(* CODESYS project 20_CS3_SQL

Project tree, tasks and I/O mapping:
  CC000xxx : 751-9401 WAGO Compact Controller 100, WAGO, order no. 751-9401, version 6.3.1.5
    application Application
      libraries: WagoSolSolutionBuilder, 1.0.0.5 (WAGO)
      task Task (cyclic, interval t#50ms, priority 15) calls PLC_PRG
      Application Template/
        ApplicationTemplateManager
          ApplicationParameters
        global variables GVL_ApplicationParameters
        program PrgRecipeHandling [ST]
        RecipeManager
          recipe definition ApplicationParameters: bLedBlinkCount : BYTE; bLedBlinkVelocity : BYTE
        text list TemplateManagerTextList
      program PLC_PRG [ST]
    Compact_Controller_100_Onboard_IO : Compact Controller 100 Onboard IO, WAGO, version 0.0.1.4
        output Application.PLC_PRG.xWD : BOOL  // X5.DO.X5.DO3
        output Application.PLC_PRG.xWD_ : BOOL  // X5.DO.X5.DO4
        unmapped channels: X12.DI, X13.PT1+/X13.PT1-, X13.PT2+/X13.PT2-, X14.AI1, X14.AI2, X5.DO, X6.AO1, X6.AO2
    Serial
      COM1 : COM1, WAGO, version 0.0.0.19
  PFC000xxx : 750-8212 PFC200, WAGO, order no. 750-8212, version 6.4.6.10
    application Application
      libraries: WagoAppRunningText, 0.0.0.1 (WAGO); WagoAppAppLED, 1.7.2.2 (WAGO); WagoSolSolutionBuilder, 1.0.0.5 (WAGO); VisuDialogs, * (System); WagoAppSQL_MySQL, 1.6.2.6 (WAGO); WagoSysErrorBase, 1.6.2.6 (WAGO); WagoSysSQLite_FR, 1.0.8.0 (WAGO_FR)
      task Task (cyclic, interval t#50ms, priority 15) calls PLC_PRG
      task TrendRecordingTask (cyclic, interval 100 ms, priority 15) calls VisuTrendStorageAccess.GlobalInstances.g_TrendRecordingManager.CyclicCall
      task VISU_TASK (cyclic, interval 100 ms, priority 15) calls VisuElems.Visu_Prg
      Application Template/
        global variables ApplicationParameters
        ApplicationTemplateManager
          ApplicationParameters
        program PrgRecipeHandling [ST]
        RecipeManager
          recipe definition ApplicationParameters: ApplicationParameters.sRunningText : STRING; ApplicationParameters.tBlinkTime01 : TIME; ApplicationParameters.tBlinkTime02 : TIME; ApplicationParameters.tBlinkTime03 : TIME; ApplicationParameters.wFunctionSelector : WORD
        text list TemplateManagerTextList
      global variables gvl_AppData
      MySQL/
      program PLC_PRG [ST]
      program PRG_MySQL [ST]
      program PRG_SQlite [ST]
      visualisation SigTrendlog
      SQlite/
      Trend Recording Manager
        SigTrendlog_Trend
      data type typSQlite_TableTest
      visualisation WSB_Example
    Kbus : Kbus, WAGO, version 2.1.0.1
        unmapped channels: K-BUS diagnostics
      _75x_16DO_1 : 75x-16DO, WAGO, version 2.0.0.13
          output wTrm1 : WORD  // _OUT
      _75x_16DO_2 : 75x-16DO, WAGO, version 2.0.0.13
          output wTrm2 : WORD  // _OUT
      _75x_16DO_3 : 75x-16DO, WAGO, version 2.0.0.13
          output wTrm3 : WORD  // _OUT
      _75x_4DI_1 : 75x-4DI, WAGO, version 2.0.0.13
          unmapped channels: _IN
    Serial
      COM1 : COM1, WAGO, version 0.0.0.19
  libraries: VisuSymbols, 4.4.0.0 (System); WagoVisuIcons, 1.1.0.8 (WAGO); WagoVisuIconsMaterialDesign, 1.0.0.2 (WAGO)
  text list GlobalTextList
*)

// PFC000xxx/Application/typSQlite_TableTest
TYPE typSQlite_TableTest :
STRUCT
	iValue			: INT;
	rValue			: REAL;
	sValue			: STRING;
	xValue			: BOOL;
END_STRUCT
END_TYPE

// PFC000xxx/Application/gvl_AppData
{attribute 'qualified_only'}
VAR_GLOBAL
	g_rSignal_SINUS				: REAL;
	g_rSignal_COSINUS			: REAL;
	g_rSignal_TRIANGLE			: REAL;
	g_rSignal_SAW				: REAL;
END_VAR

// CC000xxx/Application/Application Template/GVL_ApplicationParameters
//{attribute 'qualified_only'}
VAR_GLOBAL
	bLedBlinkCount 			: BYTE	:= 2;
	bLedBlinkVelocity 		: BYTE	:= 3;
END_VAR

// PFC000xxx/Application/Application Template/ApplicationParameters
{attribute 'qualified_only'}
VAR_GLOBAL
	// Application Parameter 1
	sRunningText: STRING := '1';
	// Application Parameter 2
	tBlinkTime01: TIME;
	// Application Parameter 3
	tBlinkTime02: TIME;
	// Application Parameter 4
	tBlinkTime03: TIME;
	// Application Parameter 5
	wFunctionSelector : WORD;		
END_VAR

// CC000xxx/Application/PLC_PRG
PROGRAM PLC_PRG
VAR
	(* cycle counter *)
	uiCnt						: UINT;
	xWD							: BOOL;
	xWD_						: BOOL;
	
END_VAR

(* cycle counter *)
uiCnt := uiCnt + 1;
xWD := uiCnt.3;
xWD_ := NOT xWD;

END_PROGRAM

// PFC000xxx/Application/PLC_PRG
PROGRAM PLC_PRG
(* **************************************************************************************** *)
(* * PROJECT INFORMATION																	*)
(* *********+***********************+****************************************************** *)
(* Author:  ¦ Stephane Rey			¦ plc acces: admin / ...								*)
(* Date:	¦ 01.07.25				¦ IP-address: 172.16.250.x/24 (dhcp)					*)
(* Version:	¦ V04.01.02.00			¦ IP-address (VPN):	10.235.0.2							*)
(* *********+*******+***************+****************************************************** *)
(* version history	¦				¦														*)
(* 01.07.25			¦ V04.01.02.00	¦ fist version											*)
(* 					¦ 				¦ CS3.5.19.07											*)
(* 					¦ 				¦														*)
(* *****************+***************+****************************************************** *)
VAR
	(* cycle counter *)
	uiCnt						: UINT;
	
	(* running text *)
	oRunningText				: WagoAppRunningText.FbRunningText;
	tRunningTextSpeed			: TIME := T#20MS;
	aRunningTextOut				: WagoAppRunningText.WLS_OUTPUTS;
	
	(* LED driver *)
	bFunctionSelectorOut		: BYTE;		
	oTOF_1						: TOF;
	oLED01						: FbAppLED_SetStatic;
	xLED01_Enable				: BOOL;
	xLED01_Error				: BOOL;
	xLED01_Valid				: BOOL;
	xLED01_Busy					: BOOL;
	oLED01_FbResult				: WagoAppAppLED.FbResult;
	eLedColor01					: WagoAppAppLED.WagoTypesAppLED.eLedColor;
	eLedColor01_				: WagoAppAppLED.WagoTypesAppLED.eLedColor;
	uiLedCount					: UINT;
	
	(* recipe management *)
	xRecipe_Read				: BOOL;
	xRecipe_Write				: BOOL;
	xRecipe_Ready				: BOOL;
	xRecipe_Busy				: BOOL;
END_VAR

(* cycle counter *)
{region 'plc-cycle-counter'}
	uiCnt := uiCnt + 1;
{endregion}

(* running text *)
{region 'running-text'}
	oRunningText(	tSpeed:= tRunningTextSpeed, 
					sText:= ApplicationParameters.sRunningText, 
					Outputs:= aRunningTextOut);
	
	(* asseign data to ourput terminals *)			
	wTrm1 := aRunningTextOut[1];	//750-1504
	wTrm2 := aRunningTextOut[2];	//750-1504
	wTrm3 := aRunningTextOut[3];	//750-1504
{endregion}

(* LED driver *)
{region 'led-driver'}
	// app selector
	CASE ApplicationParameters.wFunctionSelector OF		
		0:	// LED off
			eLedColor01:=WagoAppAppLED.WagoTypesAppLED.eLedColor.Off;
		
		1:	// LED blink yellow, sequence 1
			oTOF_1(IN:=NOT oTOF_1.Q , PT:=ApplicationParameters.tBlinkTime01);
			IF NOT oTOF_1.Q THEN
				bFunctionSelectorOut:=bFunctionSelectorOut+1;
			END_IF
			eLedColor01:=WagoAppAppLED.WagoTypesAppLED.eLedColor.Yellow;
			
		2:	// LED blink green, sequence 2
			oTOF_1(IN:=NOT oTOF_1.Q , PT:=ApplicationParameters.tBlinkTime02 );
			IF NOT oTOF_1.Q THEN
				bFunctionSelectorOut:=bFunctionSelectorOut*2;
				IF bFunctionSelectorOut=0 THEN
					bFunctionSelectorOut:=1;
				END_IF
			END_IF
			eLedColor01:=WagoAppAppLED.WagoTypesAppLED.eLedColor.Green;
			
		3:	// LED blink red, sequence 3
			oTOF_1(IN:=NOT oTOF_1.Q , PT:=ApplicationParameters.tBlinkTime03 );
			IF NOT oTOF_1.Q THEN
				bFunctionSelectorOut:=NOT bFunctionSelectorOut;
			END_IF
			eLedColor01:=WagoAppAppLED.WagoTypesAppLED.eLedColor.Red;
		ELSE
			ApplicationParameters.wFunctionSelector := 0;
	END_CASE
	
	//write new sequence management
	IF eLedColor01 <> eLedColor01_ THEN
		xLED01_Enable:=FALSE;
		uiLedCount:=uiLedCount+1;
		IF uiLedCount>10 THEN
			xLED01_Enable:=TRUE;
			eLedColor01_:=eLedColor01;
			uiLedCount:=0;
		END_IF
	END_IF
	
	// call LED driver
	oLED01(
		oStatus	=>oLED01_FbResult, 
		xEnable		:=xLED01_Enable, 
		xError		=>xLED01_Error, 
		xValid		=>xLED01_Valid, 
		xBusy		=>xLED01_Busy, 
		eLedID		:=WagoAppAppLED.eLedID.AppLED_1, 
		eLedColor	:=eLedColor01);
{endregion}	

(* recipe management *)
{region 'recipe-mngt'}
	PrgRecipeHandling(xRead:= xRecipe_Read, xWrite:= xRecipe_Write, xRecipeReady=> xRecipe_Ready, xBusy=> xRecipe_Busy);
{endregion}
	
(* application *)
{region 'application'}
	PRG_MySQL();
	PRG_SQlite();
	//ca l'air de fonctionner
{endregion}

END_PROGRAM

// CC000xxx/Application/Application Template/PrgRecipeHandling
//Program to handle the recipe parameters of the application
//{error 'Veuillez appeler ce programme dans votre programme principal ou dans une tâche pour l'activer. Supprimez ensuite cette ligne.'}
PROGRAM PrgRecipeHandling
VAR_INPUT
	xRead	: BOOL;	//Read parameters from recipe to application. (also done by tCycleTime)
	xWrite	: BOOL;	//Write parameters from application to recipe.
END_VAR
VAR_OUTPUT
	xRecipeReady	: BOOL;	//Outputs recipe parameters are ready to use in application
END_VAR
VAR
	FbRecipeApplicationParameters	: WagoSolSolutionBuilder.FbRecipeManagement;
	sApplicationParameters			: STRING:='ApplicationParameters';	//Name of the recipe definition.
	oStatusRecipeApplicationParameters	: WagoSolSolutionBuilder.WagoSysErrorBase.FbResult;
END_VAR

//call recipe manager with recipe definiction name "ApplicationParameters"
FbRecipeApplicationParameters(
	sRecipeDefinition	:= sApplicationParameters,
	tCycleTime			:= T#10S,
	xRead				:= xRead,
	xWrite				:= xWrite,
	xBusy				=> ,
	xErrorInit		=> ,
	xErrorReading	=> ,
	xErrorWriting	=> ,
	oStatus			=> oStatusRecipeApplicationParameters,
	sStatus			=> );

//handle recipe incompatibilities e.g. by adding new parameters when application was already deployed
IF FbRecipeApplicationParameters.xErrorInit OR FbRecipeApplicationParameters.xErrorReading THEN
	{IF defined (variable: GVL_RecipeManagement.g__RecipePersistencyHelper._loadType)}
	{implicit on}
	GVL_RecipeManagement.g__RecipePersistencyHelper._loadType := PersistantLoadType.LOAD_MATCHING_VARIABLES_BY_VARIABLENAME;
	{implicit off}
	FbRecipeApplicationParameters.MatchRecipe();
	{implicit on}
	GVL_RecipeManagement.g__RecipePersistencyHelper._loadType := PersistantLoadType.LOAD_TYPE_NONE;
	{implicit off}
	{END_IF}
END_IF

xRecipeReady := NOT FbRecipeApplicationParameters.xBusy;

END_PROGRAM

// PFC000xxx/Application/Application Template/PrgRecipeHandling
//Program to handle the recipe parameters of the application
//{error 'Please call this program from your main program or from a task and then remove this line'}
PROGRAM PrgRecipeHandling
VAR_INPUT
	xRead	: BOOL;	//Read parameters from recipe to application. (also done by tCycleTime)
	xWrite	: BOOL;	//Write parameters from application to recipe.
END_VAR
VAR_OUTPUT
	xRecipeReady	: BOOL;	//Outputs recipe parameters are ready to use in application
	xBusy: BOOL;
END_VAR
VAR
	FbRecipeApplicationParameters	: WagoSolSolutionBuilder.FbRecipeManagement;
	sApplicationParameters			: STRING:='ApplicationParameters';	//Name of the recipe definition.
	oStatusRecipeApplicationParameters	: WagoSolSolutionBuilder.WagoSysErrorBase.FbResult;
END_VAR

//call recipe manager with recipe definiction name "ApplicationParameters"
FbRecipeApplicationParameters(
	sRecipeDefinition	:= sApplicationParameters,
	tCycleTime			:= T#10S,
	xRead				:= xRead,
	xWrite				:= xWrite,
	xBusy				=> xBusy,
	xErrorInit		=> ,
	xErrorReading	=> ,
	xErrorWriting	=> ,
	oStatus			=> oStatusRecipeApplicationParameters,
	sStatus			=> );

//handle recipe incompatibilities e.g. by adding new parameters when application was already deployed
IF FbRecipeApplicationParameters.xErrorInit OR FbRecipeApplicationParameters.xErrorReading THEN
	{IF defined (variable: GVL_RecipeManagement.g__RecipePersistencyHelper._loadType)}
	{implicit on}
	GVL_RecipeManagement.g__RecipePersistencyHelper._loadType := PersistantLoadType.LOAD_MATCHING_VARIABLES_BY_VARIABLENAME;
	{implicit off}
	FbRecipeApplicationParameters.MatchRecipe();
	{implicit on}
	GVL_RecipeManagement.g__RecipePersistencyHelper._loadType := PersistantLoadType.LOAD_TYPE_NONE;
	{implicit off}
	{END_IF}
END_IF

xRecipeReady := NOT FbRecipeApplicationParameters.xBusy;

END_PROGRAM

// PFC000xxx/Application/PRG_MySQL
PROGRAM PRG_MySQL
(* Install a docker container within mysql DB
   ******************************************
Configure the Wago 2GB SD card as EXT4, with label “sdcard”
enable docker
ls /media/sdcard/ -l
mkdir -m 777 /media/sdcard/mysql
docker info
docker network create --driver=bridge --subnet=172.28.0.0/16 --ip-range=172.28.0.0/20 mysqlnet
docker run -d --restart always --platform=linux/arm/v7 --network mysqlnet --ip 172.28.0.10 --name mysql -p 3306:3306 -v /etc/localtime:/etc/localtime -v /media/sdcard/mysql:/var/lib/mysql -e MYSQL_ROOT_PASSWORD=password1 -e MYSQL_PASSWORD=password1 -e MYSQL_USER=user1 -e MYSQL_DATABASE=database1 biarms/mysql:5
docker ps

docker exec -it mysql sh
mysql -u root -p

show databases;
use database1;
show tables;
CREATE TABLE  myTable ( id INT AUTO_INCREMENT PRIMARY KEY, nom VARCHAR(100), prenom VARCHAR(100), created_at TIMESTAMP DEFAULT CURRENT_TIMESTAMP);
show tables;
select * from myTable;
INSERT INTO myTable (nom, prenom) VALUES ('Rey', 'Stephane');
select * from myTable;
drop myTable;
*)
VAR
	iState							: INT;
	sState							: STRING;
	aState							: ARRAY[0..c_iStateBufferSize] OF STRING;
	xMySQL_Enable					: BOOL := TRUE;
	xMySQL_Connect					: BOOL;
	xMySQL_Disconnect				: BOOL;
	xMySQL_LogData					: BOOL;
	sName							: STRING := 'CODESYS';
	sSurname						: STRING := 'Application';
	xMySQL_ClearLog					: BOOL;
	
	i								: INT;
	
	sMySQL_Host						: STRING := '127.0.0.1';
	uiMySQL_Port					: UINT := 3306;
	sMySQL_User						: STRING := 'root';
	sMySQL_Password					: STRING := 'password1';
	sMySQL_Database					: STRING := 'database1';
	
	
	(* instances *)
	// login
	oMySQL_Login					: WagoAppSQL_MySQL.FbMySql_Login;
	xMySQL_TrigConnect				: BOOL;
	xMySQL_Login_Busy				: BOOL;
	xMySQL_Login_Err				: BOOL;
	sMySQL_Login_Status				: STRING;
	xMySQL_Login_Connected			: BOOL;
	oMySQL_Login_ShowResult			: WagoSysErrorBase.FbShowResult;
	xMySQL_Login_ErrIsError			: BOOL;
	uiMySQL_Login_ErrID				: UINT;
	sMySQL_Login_ErrDesc			: STRING;
	sMySQL_Login_ErrProducer		: STRING;
	sMySQL_Login_ErrInstance		: STRING;
	eMySQL_Login_ErrSeveryty		: WagoTypes.eSeverity;
	
	// logout
	oMySQL_Logout					: WagoAppSQL_MySQL.FbMySql_Logout;
	xMySQL_TrigDisconnect			: BOOL;
	xMySQL_Logout_Busy				: BOOL;
	xMySQL_Logout_Err				: BOOL;
	sMySQL_Logout_Status			: STRING;
	oMySQL_Logout_ShowResult		: WagoSysErrorBase.FbShowResult;
	xMySQL_Logout_ErrIsError		: BOOL;
	uiMySQL_Logout_ErrID			: UINT;
	sMySQL_Logout_ErrDesc			: STRING;
	sMySQL_Logout_ErrProducer		: STRING;
	sMySQL_Logout_ErrInstance		: STRING;
	eMySQL_Logout_ErrSeveryty		: WagoTypes.eSeverity;
	
	// execute statement
	oMySQL_Execute					: WagoAppSQL_MySQL.FbMySql_Execute;
	xMySQL_TrigExecute				: BOOL;
	aMySQL_Statement				: ARRAY [0..MYSQL_SQL_UPPER_BOUND] OF STRING(MYSQL_SQL_LENGTH);
	xMySQL_Execute_Busy				: BOOL;
	xMySQL_Execute_Err				: BOOL;
	sMySQL_Execute_Status			: STRING;
	oMySQL_Execute_ShowResult		: WagoSysErrorBase.FbShowResult;
	xMySQL_Execute_ErrIsError		: BOOL;
	uiMySQL_Execute_ErrID			: UINT;
	sMySQL_Execute_ErrDesc			: STRING;
	sMySQL_Execute_ErrProducer		: STRING;
	sMySQL_Execute_ErrInstance		: STRING;
	eMySQL_Execute_ErrSeveryty		: WagoTypes.eSeverity;
	
	// send cyclicly
	oTONsend						: ton;
	tSendCycle						: TIME := T#1800S;
	
END_VAR
VAR CONSTANT
	c_iStateBufferSize				: INT := 19;
END_VAR

(* state machine *)
IF xMySQL_Enable THEN
	CASE iState OF
		0	:	// idle
				IF xMySQL_Connect THEN
					iState := 10;
				ELSIF xMySQL_Disconnect THEN
					iState := 80;
				ELSIF xMySQL_LogData THEN
					iState := 40;
				END_IF
				sState := 'MySQL idle - wait for command';
		
		10	:	// connect to DB, prepare login credentials
				oMySQL_Login.sHost:= sMySQL_Host;
				oMySQL_Login.uiPort:= uiMySQL_Port;
				oMySQL_Login.sUsername:= sMySQL_User;
				oMySQL_Login.sPassword:= sMySQL_Password;
				oMySQL_Login.sDatabase:= sMySQL_Database;
				xMySQL_TrigConnect := TRUE;
				iState := 11;
				sState := 'MySQL connect - Prepare credentials';
		
		11	:	// login
				IF NOT xMySQL_TrigConnect THEN
					IF xMySQL_Login_Err THEN
						iState := 99;
						sState := 'MySQL connect - Error';
					ELSE
						xMySQL_Connect := FALSE;
						iState := 0;
						sState := 'MySQL connect - Connected';
					END_IF
				END_IF
		
		40	:	// log data, prepare statement
				aMySQL_Statement[0] := 'INSERT INTO myTable (nom, prenom) VALUES ($'CODESYS$', $'Application$');';
				xMySQL_TrigExecute := TRUE;
				iState := 41;
				sState := 'MySQL log data - Prepare statement';
				
		41	:	//
				IF NOT xMySQL_TrigExecute THEN
					IF xMySQL_Execute_Err THEN
						iState := 99;
						sState := 'MySQL log data - send error';
					ELSE
						xMySQL_LogData := FALSE;
						iState := 0;
						sState := 'MySQL log data - send done';
					END_IF
				END_IF
				
		80	:	// disconnect from DB
				xMySQL_TrigDisconnect := TRUE;
				iState := 81;
				sState := 'MySQL disconnect - Prepare disconect command';
				
		81	:	// logout
				IF NOT xMySQL_TrigDisconnect THEN
					IF xMySQL_Logout_Err THEN
						iState := 99;
						sState := 'MySQL disconnect - Error';
					ELSE
						xMySQL_Disconnect := FALSE;
						iState := 0;
						sState := 'MySQL disconnect - Disconnected';
					END_IF
				END_IF
				
		99	: 	// Error handling
		
	ELSE
		iState := 0;
	END_CASE
ELSE
	iState := 0;
END_IF

(* instances *)
{region 'call-instances'}
	// login
	oMySQL_Login(
		xTrigger:= xMySQL_TrigConnect, 
		xBusy=> xMySQL_Login_Busy, 
		xError=> xMySQL_Login_Err, 
		oStatus=> , 
		sStatus=> sMySQL_Login_Status, 
		xConnected=> xMySQL_Login_Connected);
	oMySQL_Login_ShowResult(
		IResult:= oMySQL_Login.oStatus, 
		xIsError=> xMySQL_Login_ErrIsError, 
		uiID=> uiMySQL_Login_ErrID, 
		sDescription=> sMySQL_Login_ErrDesc, 
		sProducer=> sMySQL_Login_ErrProducer, 
		sInstance=> sMySQL_Login_ErrInstance, 
		eSeverity=> eMySQL_Login_ErrSeveryty);
		
	//logout
	oMySQL_Logout(
		xTrigger:= xMySQL_TrigDisconnect, 
		xBusy=> xMySQL_Logout_Busy, 
		xError=> xMySQL_Logout_Err, 
		oStatus=> , 
		sStatus=> sMySQL_Logout_Status);
	oMySQL_Logout_ShowResult(
		IResult:= oMySQL_Logout.oStatus, 
		xIsError=> xMySQL_Logout_ErrIsError, 
		uiID=> uiMySQL_Logout_ErrID, 
		sDescription=> sMySQL_Logout_ErrDesc, 
		sProducer=> sMySQL_Logout_ErrProducer, 
		sInstance=> sMySQL_Logout_ErrInstance, 
		eSeverity=> eMySQL_Logout_ErrSeveryty);
	
	//execute statement
	oMySQL_Execute(
		aSqlCommand:= aMySQL_Statement, 
		xTrigger:= xMySQL_TrigExecute, 
		xBusy=> xMySQL_Execute_Busy, 
		xError=> xMySQL_Execute_Err, 
		oStatus=> , 
		sStatus=> sMySQL_Execute_Status);
	oMySQL_Execute_ShowResult(
		IResult:= oMySQL_Execute.oStatus, 
		xIsError=> xMySQL_Execute_ErrIsError, 
		uiID=> uiMySQL_Execute_ErrID, 
		sDescription=> sMySQL_Execute_ErrDesc, 
		sProducer=> sMySQL_Execute_ErrProducer, 
		sInstance=> sMySQL_Execute_ErrInstance, 
		eSeverity=> eMySQL_Execute_ErrSeveryty);
		
	// send cyclicly
	oTONsend(IN:= NOT oTONsend.Q AND xMySQL_Login_Connected, PT:= tSendCycle, Q=> , ET=> );
	IF oTONsend.Q THEN
		xMySQL_TrigExecute := TRUE;
	END_IF
{endregion}
	
{region 'magt-state-fuffer'}
	IF sState <> aState[0] THEN 
		FOR i:= c_iStateBufferSize TO 1 BY -1 DO
			aState[i] := aState[i-1];
		END_FOR
	END_IF
	aState[0] := sState;
	IF xMySQL_ClearLog	THEN
		FOR i:= 0 TO c_iStateBufferSize DO
			aState[i] := '';
		END_FOR
		xMySQL_ClearLog := FALSE;
	END_IF
{endregion}

END_PROGRAM

// PFC000xxx/Application/PRG_SQlite
PROGRAM PRG_SQlite
VAR
	iState							: INT;
	sState							: STRING;
	aState							: ARRAY[0..c_iStateBufferSize] OF STRING;
	xSQlite_Enable					: BOOL := TRUE;
	xSQlite_Connect					: BOOL;
	xSQlite_Disconnect				: BOOL;
	xSQlite_CreateTab				: BOOL;
	xSQlite_LogData					: BOOL;
	xSQlite_ReadData				: BOOL;
	xSQlite_ClearLog				: BOOL;
	
	i								: INT;
	
	sSQlite_DBpath					: STRING := '/media/sd/sqlite';
	sSQlite_Filename				: STRING := 'db1';
	xSQlite_OnSDcard				: BOOL := FALSE;
	xSQlite_ClassicPath				: BOOL := FALSE;
	
	sSQL_Statement					: STRING(255);
	iValue							: INT := 12345;
	rValue							: REAL := 3.14159;
	sValue							: STRING := 'hello';
	xValue							: BOOL;
	
	aTableValues					: ARRAY[1..c_iMaxTableSize] OF typSQlite_TableTest;
	
	(* instances *)
	oSQlite							: WagoSysSQLite_FR.FbSQLite;
	xSQlite_BeginTransac 			: BOOL;
	xSQlite_Err						: BOOL;
	sSQlite_Status					: STRING;
	xSQlite_DBexist					: BOOL;
	
	
	
END_VAR
VAR CONSTANT
	c_iStateBufferSize				: INT := 19;
	c_iMaxTableSize					: INT := 99;
END_VAR

(* state machine *)
IF xSQlite_Enable THEN
	CASE iState OF
		0	:	// idle
				xSQlite_ClearLog := xSQlite_ClearLog;
				IF xSQlite_Connect THEN
					iState := 10;
				ELSIF xSQlite_Disconnect THEN
					iState := 80;
				ELSIF xSQlite_CreateTab THEN
					iState := 20;
				ELSIF xSQlite_LogData THEN
					iState := 40;
				ELSIF xSQlite_ReadData THEN
					iState := 50;
				END_IF
				sState := 'SQlite idle - wait for command';
				
		10	:	// open tDB
				IF oSQlite.open(sPath := sSQlite_DBpath, sFilename := sSQlite_Filename, xOnSDCard := xSQlite_OnSDcard, xClassicPath := xSQlite_ClassicPath, xBeginTransaction := xSQlite_BeginTransac, xError => xSQlite_Err, sStatus => sSQlite_Status, xDbExists => xSQlite_DBexist) THEN
					IF 	xSQlite_Err THEN
						iState := 99;
						sState := 'SQlite open DB - open error';
					ELSE
						iState := 11;
						sState := 'SQlite open DB - openning DB';
					END_IF
				END_IF
		
		11	:	// log
				iState := 12;
				sState := sSQlite_Status;
						
		12	:	// DB is open
				xSQlite_Connect := FALSE;
				iState := 0;
				sState := 'SQlite open DB - DB is open';
				
		20	:	// create table
				//sSQL_Statement := 'CREATE TABLE IF NOT EXISTS table_test(id INTEGER PRIMARY KEY AUTOINCREMENT, Val_1 INTEGER, Val_2 REAL, Val_3 TEXT, Val_4 INTEGER)';
				sSQL_Statement := 'CREATE TABLE IF NOT EXISTS table_test(Val_1 INTEGER, Val_2 REAL, Val_3 TEXT, Val_4 INTEGER)';
				oSQlite.executeSQLCommand(
					sSQLrequest := sSQL_Statement,
					xError => xSQlite_Err,
					sStatus => sSQlite_Status);
				iState := 21;
				sState := 'SQlite create table - create';
				
		21	:	// finalize
				IF xSQlite_Err THEN
					iState := 99;
					sState := 'SQlite create table - error';
				ELSE
					oSQlite.finalize();
					iState := 22;
					sState := sSQlite_Status;					
				END_IF
				xSQlite_LogData := FALSE;
				
		22	:	// create table, done
				xSQlite_CreateTab := FALSE;
				iState := 0;
				sState := 'SQlite create table - done';
				
		40	:	// log data, prepare statement
				sSQL_Statement := 'INSERT INTO table_test VALUES (?,?,?,?)';	//(iValue INTEGER, sValue TEXT, rValue REAL, diValue DINT, lrValue DOUBLE, liValue INTEGER, xValue INTEGER)
				oSQlite.insertData4(
					sSQLrequest := sSQL_Statement,
					value1 := iValue,
					value2 := rValue,
					value3 := sValue,
					value4 := xValue,
					xError => xSQlite_Err,
					sStatus => sSQlite_Status);
				iState := 41;
				sState := 'SQlite log data - write';
				
		41	:	// finalize
				IF xSQlite_Err THEN
					iState := 99;
					sState := 'SQlite log data - error';
				ELSE
					oSQlite.finalize();
					iState := 42;
					sState := sSQlite_Status;					
				END_IF
				
		42	:	// log data, done				
				xSQlite_LogData := FALSE;			
				iState := 0;
				sState := 'SQlite log data - done';	
				
		50	:	// read data, prepare statement
				sSQL_Statement := 'SELECT * FROM table_test';
				FOR i:= 1 TO c_iMaxTableSize DO
					IF NOT oSQlite.getData4(
						sSQLrequest := sSQL_Statement,
						value1 := aTableValues[i].iValue,
						value2 := aTableValues[i].rValue,
						value3 := aTableValues[i].sValue,
						value4 := aTableValues[i].xValue,
						xError => xSQlite_Err,
						sStatus => sSQlite_Status) THEN
							EXIT; //If no data available or error, exit from the loop
					END_IF
				END_FOR
				oSQlite.finalize();
				
				xSQlite_ReadData := FALSE;
				iState := 0;
				
		80	:	// close DB
				IF oSQlite.close(xCommitTransaction := TRUE, xError := xSQlite_Err, sStatus := sSQlite_Status) THEN
					iState := 81;
					sState := 'SQlite close DB - closing DB';					
				END_IF
				
		81	:	// log
				iState := 82;
				sState := sSQlite_Status;
				
		82	:	// DB is close
				xSQlite_Disconnect := FALSE;
				iState := 0;
				sState := 'SQlite close DB - DB is closed';				
		
		99	:	// error handling
				sState := sSQlite_Status;
	ELSE
		iState := 0;
	END_CASE
ELSE
	xSQlite_Connect := FALSE;
	xSQlite_Disconnect := FALSE;
	xSQlite_CreateTab := FALSE;
	xSQlite_LogData := FALSE;
	xSQlite_ReadData := FALSE;
	iState := 0;
END_IF

{region 'magt-state-fuffer'}
	IF sState <> aState[0] THEN 
		FOR i:= c_iStateBufferSize TO 1 BY -1 DO
			aState[i] := aState[i-1];
		END_FOR
	END_IF
	aState[0] := sState;
	IF xSQlite_ClearLog	THEN
		FOR i:= 0 TO c_iStateBufferSize DO
			aState[i] := '';
		END_FOR
		xSQlite_ClearLog := FALSE;
	END_IF
{endregion}

END_PROGRAM

// PFC000xxx/Application/SigTrendlog
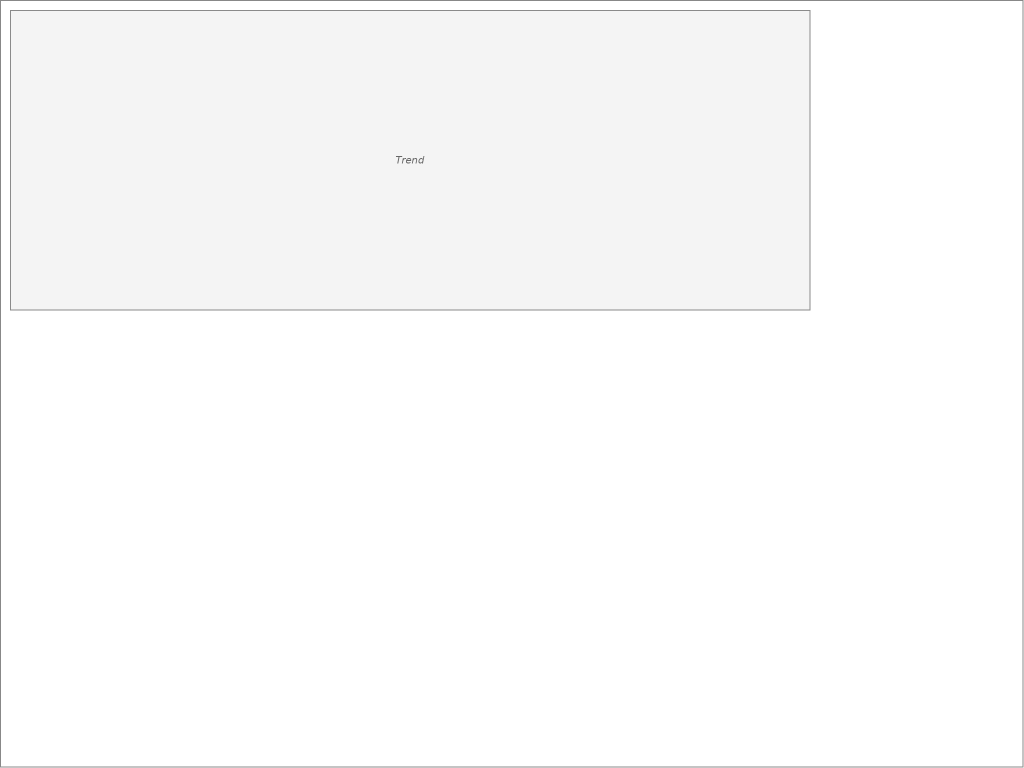
VISUALIZATION SigTrendlog  // 1024x768
    Trend (10,10 800x300)
        p758368661: dd.MM.yyyy
        p2423372160: HH:mm:ss:ms
        p2833066001: SigTrendlog_Trend
END_VISUALIZATION

// PFC000xxx/Application/WSB_Example
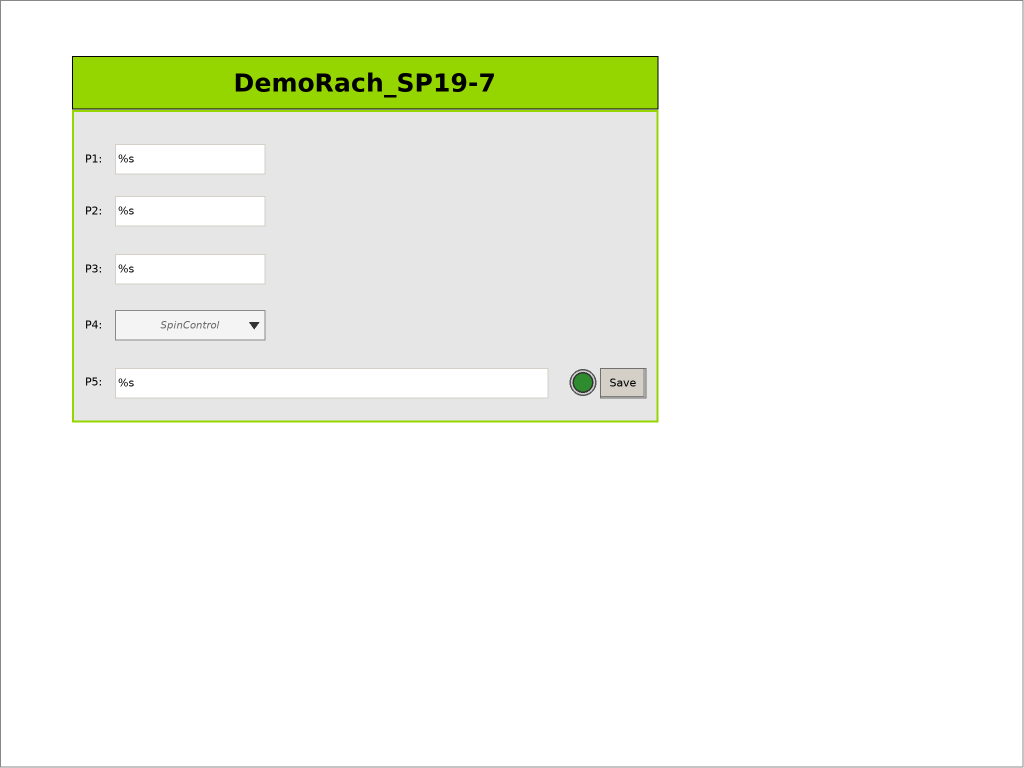
VISUALIZATION WSB_Example  // 1024x768
    Rectangle (72,110 586x312)
    Rectangle (72,56 586x53), "DemoRach_SP19-7", tooltip "Training WAGO Solution Builder"
    Textfield (115,144 150x30), "%s", text variable: ApplicationParameters.tBlinkTime01
    Textfield (115,254 150x30), "%s", text variable: ApplicationParameters.tBlinkTime03
    Textfield (115,368 433x30), "%s", text variable: ApplicationParameters.sRunningText
        OnMouseDown: write the text variable via Default
    SpinControl (115,310 150x30), variable: ApplicationParameters.wFunctionSelector
    Lamp1 (567,367 32x31), variable: PrgRecipeHandling.xBusy, style: Lamp-Lamp1-Green
    Label (73,254 32x30), "P3:"
    Label (73,367 32x30), "P5:"
    Label (73,310 32x30), "P4:"
    Label (73,144 32x30), "P1:"
    Button (600,368 46x30), "Save"
        OnMouseDown:  ToggleVariable=PrgRecipeHandling.xWrite
    Textfield (115,196 150x30), "%s", text variable: ApplicationParameters.tBlinkTime02
    Label (73,196 32x30), "P2:"
END_VISUALIZATION

(* text list TemplateManagerTextList (id | default)
   | 
  ApplicationTemplateManager.TemplateDescription | Description of DemoRack_SP19-7 / PFC200 application
  ApplicationTemplateManager.TemplateTitle | DemoRack_V4-1-2-1_SP19-7_CC-FW28 *)

(* text list TemplateManagerTextList (id | default)
   | 
  ApplicationTemplateManager.TemplateTitle | DemoRack_V4-1-2-1_SP19-7_PFC-FW28
  ApplicationTemplateManager.TemplateDescription | Description of DemoRack_SP19-7 / PFC200 application *)
